FUNCTION Convert_USINT_TO_WORD : BOOL
VAR_INPUT
	in : USINT;
	out : REFERENCE TO WORD;
END_VAR
VAR
	converted : WORD;
END_VAR

converted := USINT_TO_WORD(in);

IF (WORD_TO_USINT(converted) <> in) THEN
	RETURN;
END_IF

out := converted;
Convert_USINT_TO_WORD := TRUE;

END_FUNCTION

(* stored: Version 1.1.0.1, ProductVersion 3.1.4024.12
   POU Convert_USINT_TO_WORD: Id {f0e92edd-479c-4f6c-8f4c-4ae2d3eb4c00}, SpecialFunc None *)
